Yaskawa INFORM job: SET_TCPON.JBI

/JOB
//NAME SET_TCPON
///FOLDERNAME TWINCAT_KOMMUNIKATION
//POS
///NPOS 0,0,0,0,0,0
//ALIAS
///LVARS 0,1,0,0,0,0,0,0
LI000 TCP_NR
//ARGINFO
///ARGTYPE I,,,,,,,
///COMMENT
TCP_NR







//INST
///DATE 2021/04/27 10:40
///ATTR SC,RW
///LVARS 0,1,0,0,0,0,0,0
NOP
GETARG TCP_NR IARG#(1)
SETREG MREG#(67) TCP_NR
END
